Fanuc KAREL source: kc00028.KL

-- PROVISIONAL review KL for V940-1; original PC SHA256 17896e0c247b54878c1142eb12c466bc03a1eefc2c673c1e1f72037b2b619128
-- Incomplete behavior may be omitted. Consult companion uncertainty JSON. Do not deploy.
PROGRAM KC00028
%NOLOCKGROUP
BEGIN
  -- V9_ZERO_TABLE_METADATA_HINT layout=0002_ascii; no indexed target words; source/name/runtime held
  -- UNRESOLVED_PC offsets 5-93; opcodes 27,22,1C,22,1C,22,1C,22,1C,22,22,22,22,1C,22,31
  -- UNRESOLVED_PC offsets 98-102; opcodes 7F
END KC00028
